(* Logix 5000 project; controller STAT 1756-L72 rev 20.12; software revision 20.04; part 10 of 34 *)
(* tags used below, declared in another part *)
   B3 : DINT[256];
   CDRO1 : REAL;
   CDRO2 : REAL;
   CDRO3 : REAL;
   COND1_EAURECYCL : REAL;
   COND2_OSMOS : DINT;
   COND3 : REAL;
   COND4 : REAL;
   COND7 : REAL;
   cond_6 : REAL;
   F8 : REAL[256];
   FLW_CO1 : REAL;
   FLW_CO2 : REAL;
   FLW_CO3 : REAL;
   FLW_EAU_VILLE : REAL;
   FLW_PO1 : REAL;
   FLW_PO2 : REAL;
   FLW_PO3 : REAL;
   hard : REAL;
   I20_000 : ALIAS FOR I20[0];
   I20_001 : ALIAS FOR I20[1];
   I20_002 : ALIAS FOR I20[2];
   I20_003 : ALIAS FOR I20[3];
   I20_004 : ALIAS FOR I20[4];
   I20_005 : ALIAS FOR I20[5];
   I20_006 : ALIAS FOR I20[6];
   I20_007 : ALIAS FOR I20[7];
   I21_000 : ALIAS FOR I21[0];
   I21_001 : ALIAS FOR I21[1];
   I21_002 : ALIAS FOR I21[2];
   I21_003 : ALIAS FOR I21[3];
   I21_004 : ALIAS FOR I21[4];
   I21_005 : ALIAS FOR I21[5];
   I21_006 : ALIAS FOR I21[6];
   I22_000 : ALIAS FOR I22[0];
   I22_001 : ALIAS FOR I22[1];
   I22_002 : ALIAS FOR I22[2];
   I22_003 : ALIAS FOR I22[3];
   I22_004 : ALIAS FOR I22[4];
   I22_005 : ALIAS FOR I22[5];
   I22_006 : ALIAS FOR I22[6];
   I22_007 : ALIAS FOR I22[7];
   I23_000 : ALIAS FOR I23[0];
   I23_001 : DINT;
   I23_003 : ALIAS FOR I23[3];
   I23_004 : ALIAS FOR I23[4];
   I23_005 : ALIAS FOR I23[5];
   I23_006 : ALIAS FOR I23[6];
   I24_000 : ALIAS FOR I24[0];
   I25_000 : ALIAS FOR I25[0];
   I25_001 : ALIAS FOR I25[1];
   I25_002 : ALIAS FOR I25[2];
   I25_003 : ALIAS FOR I25[3];
   I25_005 : ALIAS FOR I25[5];
   I25_006 : ALIAS FOR I25[6];
   I25_007 : ALIAS FOR I25[7];
   I26_000 : ALIAS FOR I26[0];
   I26_001 : ALIAS FOR I26[1];
   I26_002 : ALIAS FOR I26[2];
   int_flw_put3 : integrat;
   KRK_K1 : REAL;
   LDN_L1 : DINT;
   LVL_AZ : REAL;
   LVL_LUS2_ACIDE : REAL;
   LVL_LUS3_NAOH : REAL;
   LVL_PRETRAITEMENT : REAL;
   LVL_PUISARD_IBT : DINT;
   LVL_PUISARD_L4 : REAL;
   LVL_ZOUT : REAL;
   MW : BOOL;
   N12 : DINT[230];
   N12_110 : REAL;
   N12_14 : REAL;
   N12_38 : REAL;
   N12_44 : REAL;
   N19 : DINT[80];
   N23 : DINT[80];
   N26 : DINT[256];
   N7 : DINT[255];
   N7_70 : REAL;
   N7_72 : REAL;
   O22_000_Bit04 : ALIAS FOR O22[0].4;
   PH11 : REAL;
   PH12 : REAL;
   PH2_PRETRAIT : REAL;
   Q2 : REAL;
   Q3 : REAL;
   Q4 : REAL;
   QUAT_Q1 : REAL;
   S_FLOW_PUT_1 : DINT;
   S_FLOW_PUT_2 : DINT;
   S_FLOW_VENTURI : DINT;
   S_LVL_VIJVER : REAL;
   scp_110 : SCP;
   scp_cdro1 : SCP;
   scp_cdro2 : SCP;
   scp_cdro3 : SCP;
   scp_COND1 : SCP;
   scp_COND2_OS : SCP;
   scp_COND3 : SCP;
   scp_COND4 : SCP;
   scp_COND7 : SCP;
   scp_cond_venturi : SCP;
   scp_EAU_VILLE : SCP;
   scp_FLW_CO1 : SCP;
   scp_FLW_CO2 : SCP;
   scp_FLW_CO3 : SCP;
   scp_FLW_PO1 : SCP;
   scp_FLW_PO2 : SCP;
   scp_FLW_PO3 : SCP;
   scp_flw_put1 : SCP;
   scp_flw_put2 : SCP;
   scp_flw_put3 : SCP;
   scp_FLW_Q3 : SCP;
   scp_flw_venturi : SCP;
   scp_hard : SCP;
   scp_KR_1 : SCP;
   scp_LDN_1 : SCP;
   scp_LUS2 : SCP;
   scp_LUS3 : SCP;
   scp_LVL_AZ : SCP;
   scp_lvl_l4 : SCP;
   scp_LVL_PRET : SCP;
   scp_LVL_PUIS : SCP;
   scp_LVL_PUIS_L4 : SCP;
   scp_lvl_vijver : SCP;
   scp_LVL_ZOUT : SCP;
   scp_N12_14 : SCP;
   scp_N12_38 : SCP;
   scp_N12_44 : SCP;
   scp_N7_70 : SCP;
   scp_N7_72 : SCP;
   scp_PH11 : SCP;
   scp_PH12 : SCP;
   scp_PH2 : SCP;
   scp_ph_venturi : SCP;
   scp_Q2 : SCP;
   scp_Q4 : SCP;
   scp_QUAT_Q1 : SCP;
   scp_t_venturi : SCP;
   scpcond_6 : SCP;
(* ibt, continued *)

ROUTINE _13_ANALOG   (* ladder *)
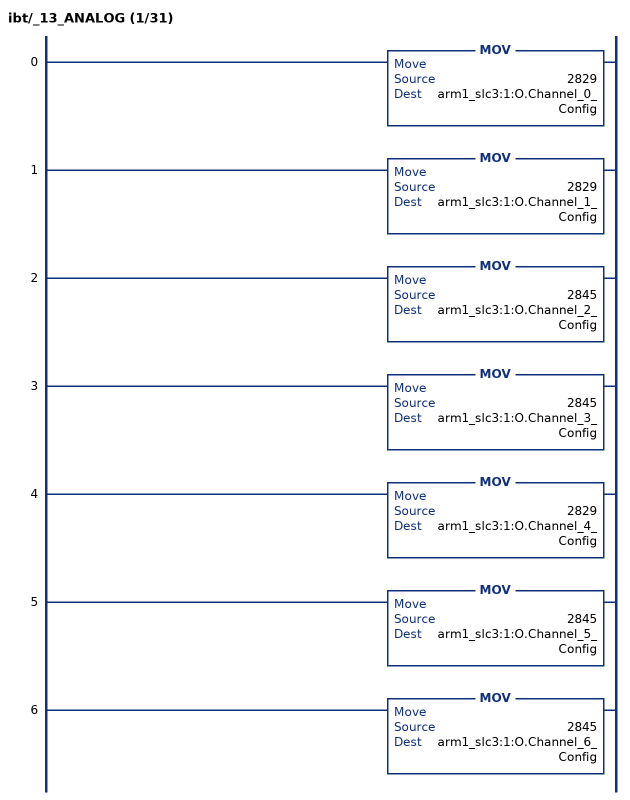
   0: MOV(2829,arm1_slc3:1:O.Channel_0_Config);
   1: MOV(2829,arm1_slc3:1:O.Channel_1_Config);
   2: MOV(2845,arm1_slc3:1:O.Channel_2_Config);
   3: MOV(2845,arm1_slc3:1:O.Channel_3_Config);
   4: MOV(2829,arm1_slc3:1:O.Channel_4_Config);
   5: MOV(2845,arm1_slc3:1:O.Channel_5_Config);
   6: MOV(2845,arm1_slc3:1:O.Channel_6_Config);
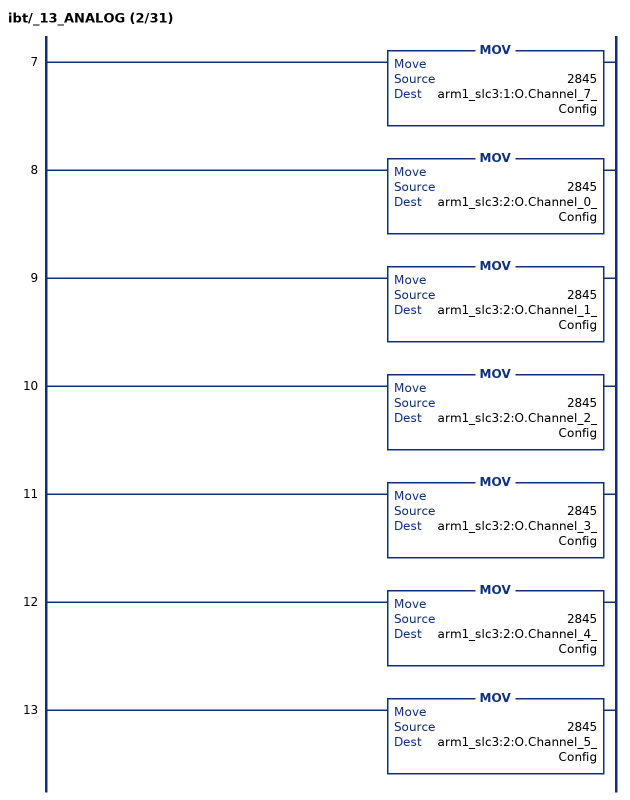
   7: MOV(2845,arm1_slc3:1:O.Channel_7_Config);
   8: MOV(2845,arm1_slc3:2:O.Channel_0_Config);
   9: MOV(2845,arm1_slc3:2:O.Channel_1_Config);
   10: MOV(2845,arm1_slc3:2:O.Channel_2_Config);
   11: MOV(2845,arm1_slc3:2:O.Channel_3_Config);
   12: MOV(2845,arm1_slc3:2:O.Channel_4_Config);
   13: MOV(2845,arm1_slc3:2:O.Channel_5_Config);
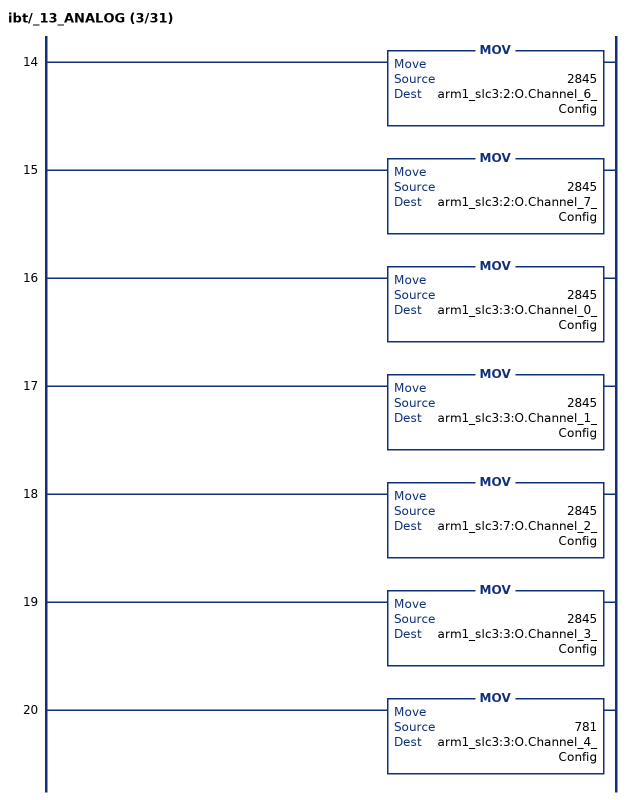
   14: MOV(2845,arm1_slc3:2:O.Channel_6_Config);
   15: MOV(2845,arm1_slc3:2:O.Channel_7_Config);
   16: MOV(2845,arm1_slc3:3:O.Channel_0_Config);
   17: MOV(2845,arm1_slc3:3:O.Channel_1_Config);
   18: MOV(2845,arm1_slc3:7:O.Channel_2_Config);
   19: MOV(2845,arm1_slc3:3:O.Channel_3_Config);
   20: MOV(781,arm1_slc3:3:O.Channel_4_Config);
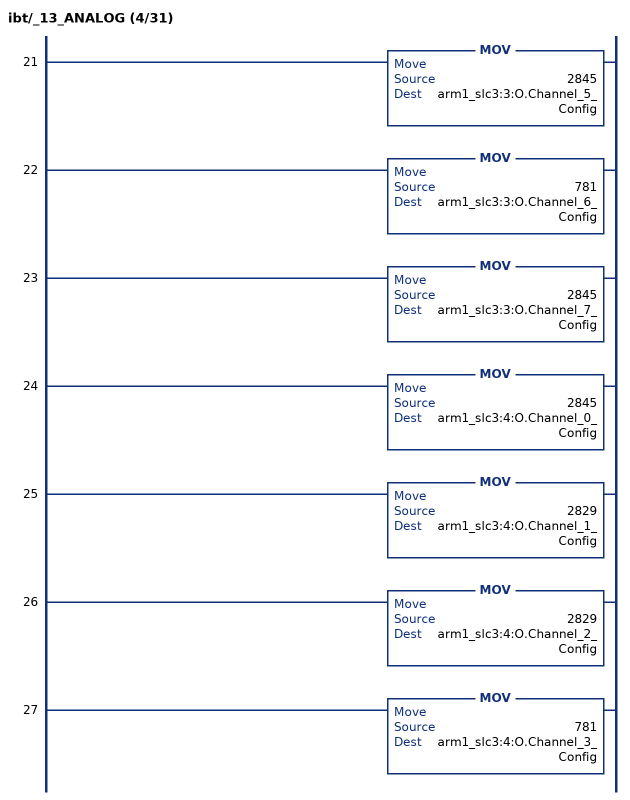
   21: MOV(2845,arm1_slc3:3:O.Channel_5_Config);
   22: MOV(781,arm1_slc3:3:O.Channel_6_Config);
   23: MOV(2845,arm1_slc3:3:O.Channel_7_Config);
   24: MOV(2845,arm1_slc3:4:O.Channel_0_Config);
   25: MOV(2829,arm1_slc3:4:O.Channel_1_Config);
   26: MOV(2829,arm1_slc3:4:O.Channel_2_Config);
   27: MOV(781,arm1_slc3:4:O.Channel_3_Config);
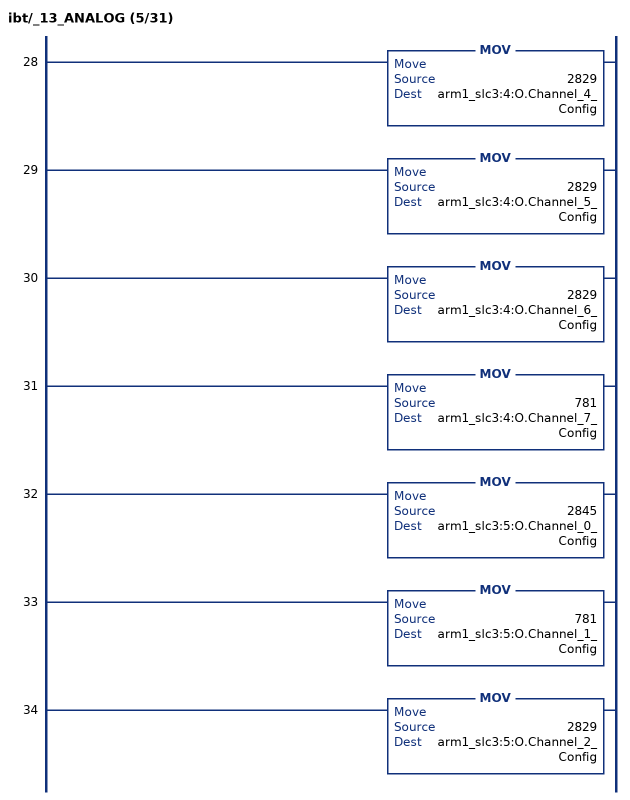
   28: MOV(2829,arm1_slc3:4:O.Channel_4_Config);
   29: MOV(2829,arm1_slc3:4:O.Channel_5_Config);
   30: MOV(2829,arm1_slc3:4:O.Channel_6_Config);
   31: MOV(781,arm1_slc3:4:O.Channel_7_Config);
   32: MOV(2845,arm1_slc3:5:O.Channel_0_Config);
   33: MOV(781,arm1_slc3:5:O.Channel_1_Config);
   34: MOV(2829,arm1_slc3:5:O.Channel_2_Config);
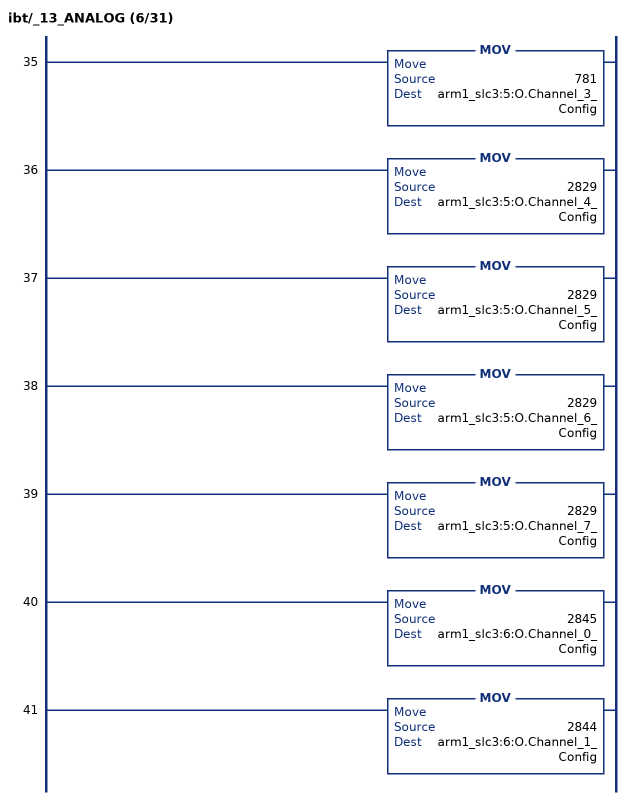
   35: MOV(781,arm1_slc3:5:O.Channel_3_Config);
   36: MOV(2829,arm1_slc3:5:O.Channel_4_Config);
   37: MOV(2829,arm1_slc3:5:O.Channel_5_Config);
   38: MOV(2829,arm1_slc3:5:O.Channel_6_Config);
   39: MOV(2829,arm1_slc3:5:O.Channel_7_Config);
   40: MOV(2845,arm1_slc3:6:O.Channel_0_Config);
   41: MOV(2844,arm1_slc3:6:O.Channel_1_Config);
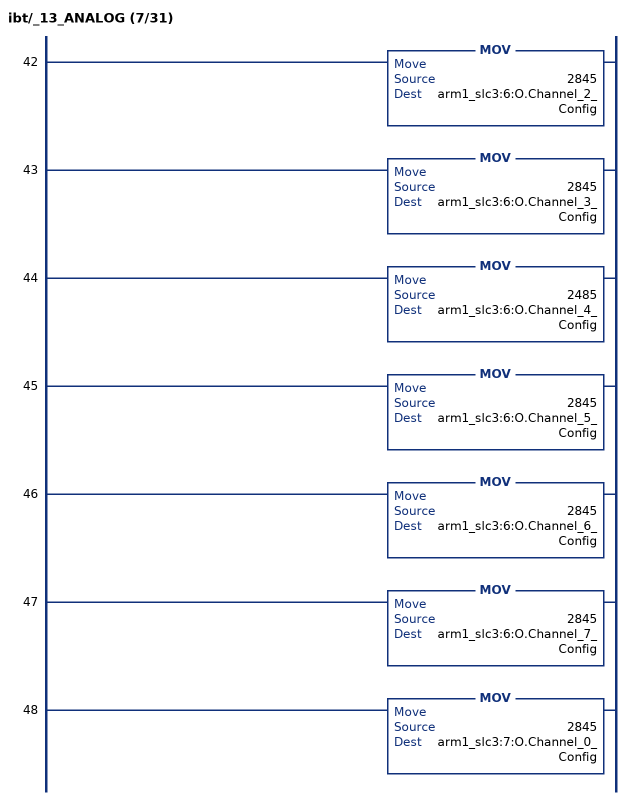
   42: MOV(2845,arm1_slc3:6:O.Channel_2_Config);
   43: MOV(2845,arm1_slc3:6:O.Channel_3_Config);
   44: MOV(2485,arm1_slc3:6:O.Channel_4_Config);
   45: MOV(2845,arm1_slc3:6:O.Channel_5_Config);
   46: MOV(2845,arm1_slc3:6:O.Channel_6_Config);
   47: MOV(2845,arm1_slc3:6:O.Channel_7_Config);
   48: MOV(2845,arm1_slc3:7:O.Channel_0_Config);
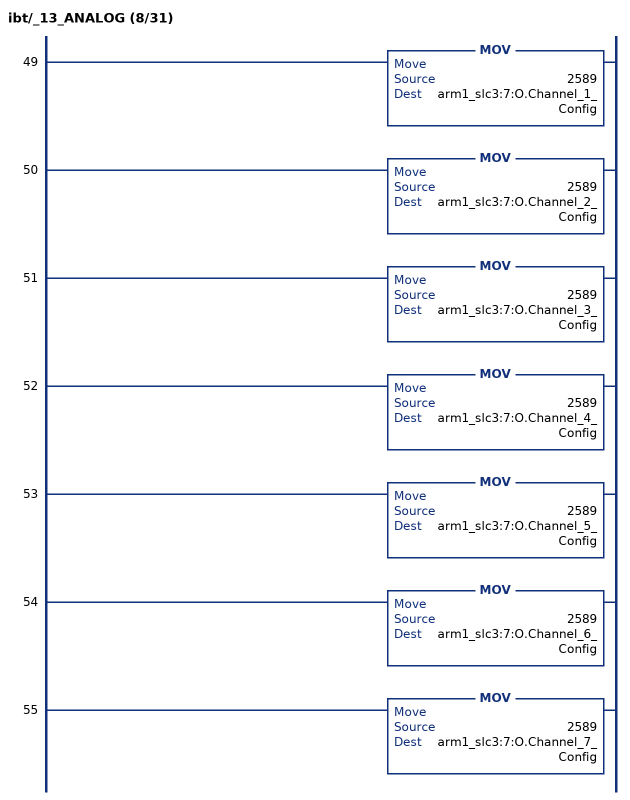
   49: MOV(2589,arm1_slc3:7:O.Channel_1_Config);
   50: MOV(2589,arm1_slc3:7:O.Channel_2_Config);
   51: MOV(2589,arm1_slc3:7:O.Channel_3_Config);
   52: MOV(2589,arm1_slc3:7:O.Channel_4_Config);
   53: MOV(2589,arm1_slc3:7:O.Channel_5_Config);
   54: MOV(2589,arm1_slc3:7:O.Channel_6_Config);
   55: MOV(2589,arm1_slc3:7:O.Channel_7_Config);
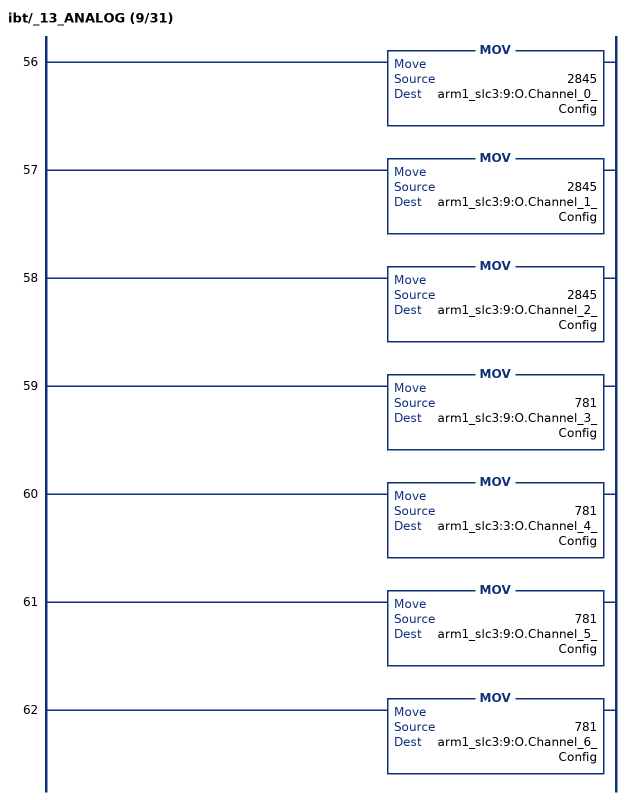
   56: MOV(2845,arm1_slc3:9:O.Channel_0_Config);
   57: MOV(2845,arm1_slc3:9:O.Channel_1_Config);
   58: MOV(2845,arm1_slc3:9:O.Channel_2_Config);
   59: MOV(781,arm1_slc3:9:O.Channel_3_Config);
   60: MOV(781,arm1_slc3:3:O.Channel_4_Config);
   61: MOV(781,arm1_slc3:9:O.Channel_5_Config);
   62: MOV(781,arm1_slc3:9:O.Channel_6_Config);
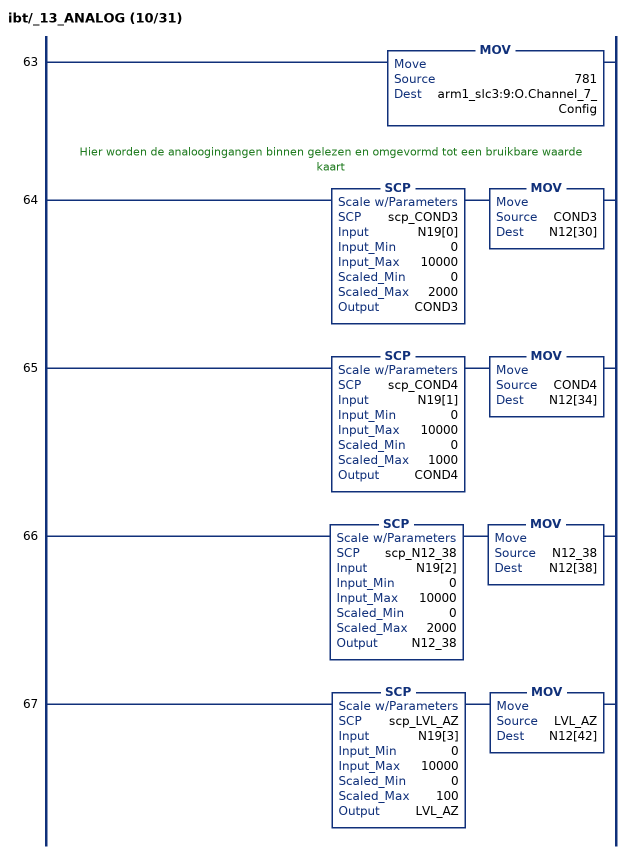
   63: MOV(781,arm1_slc3:9:O.Channel_7_Config);
   // Hier worden de analoogingangen binnen gelezen en omgevormd tot een bruikbare waarde kaart
   64: SCP(scp_COND3,N19[0],0,10000,0,2000,COND3)MOV(COND3,N12[30]);
   65: SCP(scp_COND4,N19[1],0,10000,0,1000,COND4)MOV(COND4,N12[34]);
   66: SCP(scp_N12_38,N19[2],0,10000,0,2000,N12_38)MOV(N12_38,N12[38]);
   67: SCP(scp_LVL_AZ,N19[3],0,10000,0,100,LVL_AZ)MOV(LVL_AZ,N12[42]);
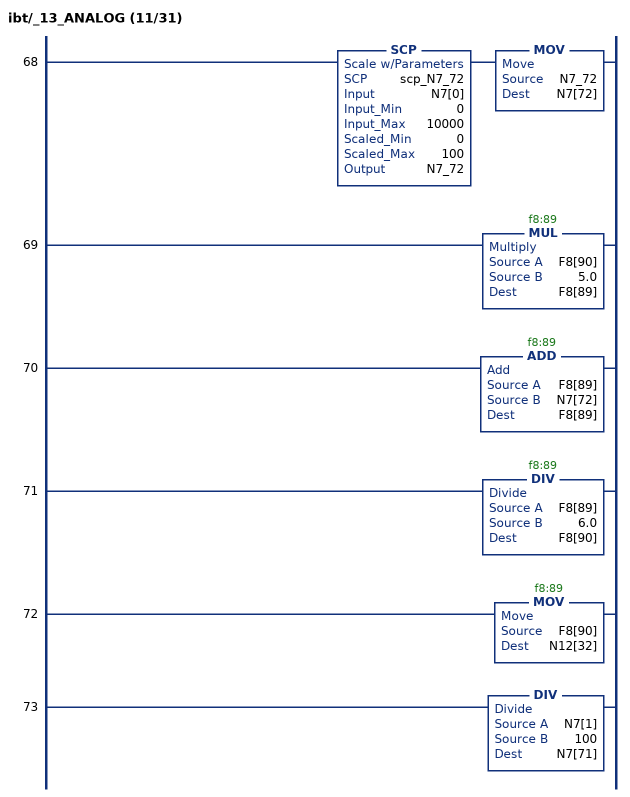
   68: SCP(scp_N7_72,N7[0],0,10000,0,100,N7_72)MOV(N7_72,N7[72]);
   69: MUL(F8[90],5.0,F8[89]);
   70: ADD(F8[89],N7[72],F8[89]);
   71: DIV(F8[89],6.0,F8[90]);
   72: MOV(F8[90],N12[32]);
   73: DIV(N7[1],100,N7[71]);
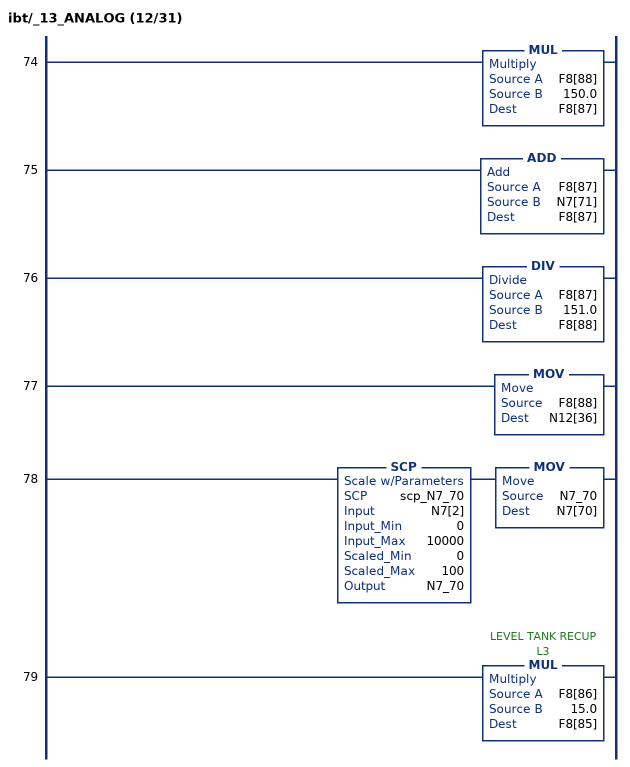
   74: MUL(F8[88],150.0,F8[87]);
   75: ADD(F8[87],N7[71],F8[87]);
   76: DIV(F8[87],151.0,F8[88]);
   77: MOV(F8[88],N12[36]);
   78: SCP(scp_N7_70,N7[2],0,10000,0,100,N7_70)MOV(N7_70,N7[70]);
   79: MUL(F8[86],15.0,F8[85]);
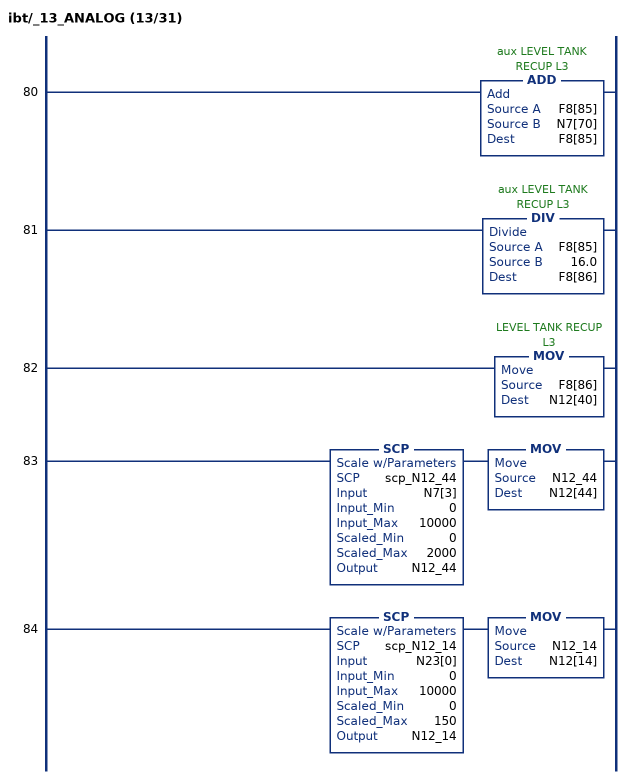
   80: ADD(F8[85],N7[70],F8[85]);
   81: DIV(F8[85],16.0,F8[86]);
   82: MOV(F8[86],N12[40]);
   83: SCP(scp_N12_44,N7[3],0,10000,0,2000,N12_44)MOV(N12_44,N12[44]);
   84: SCP(scp_N12_14,N23[0],0,10000,0,150,N12_14)MOV(N12_14,N12[14]);
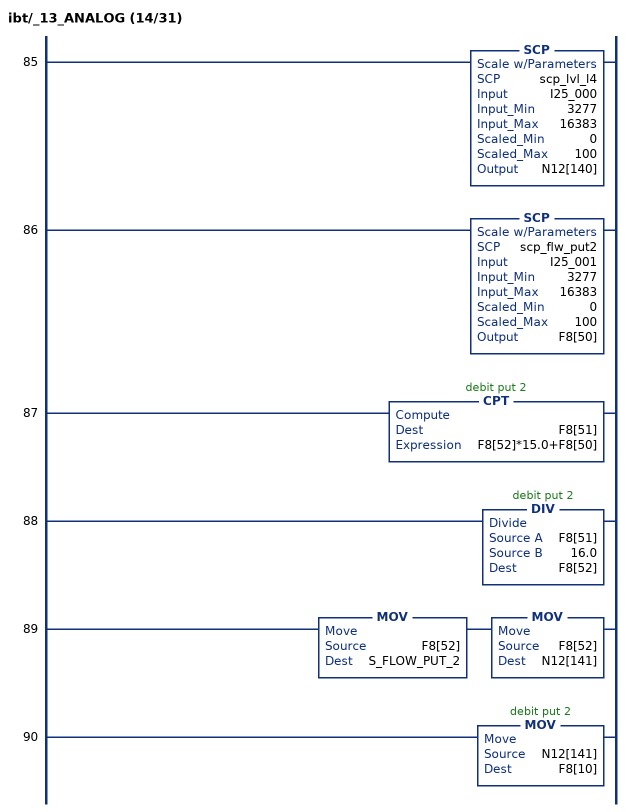
   85: SCP(scp_lvl_l4,I25_000,3277,16383,0,100,N12[140]);
   86: SCP(scp_flw_put2,I25_001,3277,16383,0,100,F8[50]);
   87: CPT(F8[51],F8[52]*15.0+F8[50]);
   88: DIV(F8[51],16.0,F8[52]);
   89: MOV(F8[52],S_FLOW_PUT_2)MOV(F8[52],N12[141]);
   90: MOV(N12[141],F8[10]);
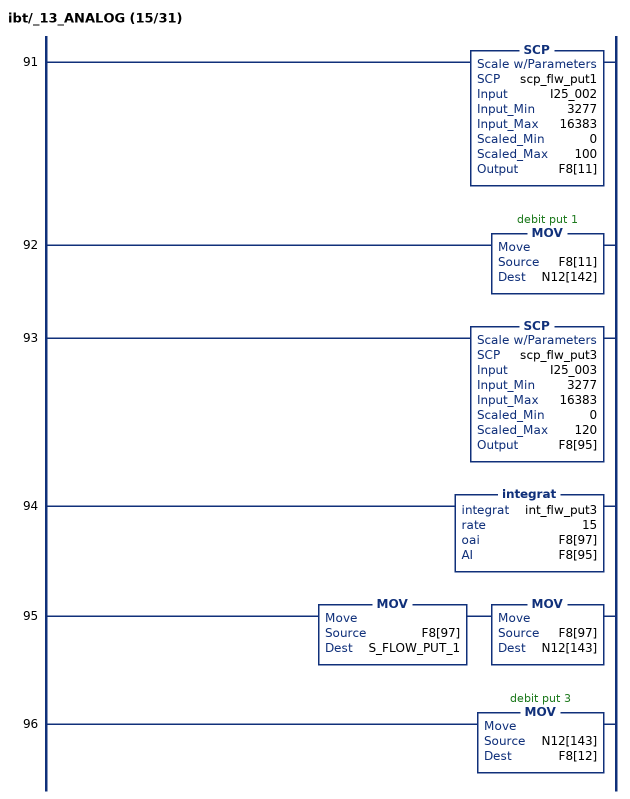
   91: SCP(scp_flw_put1,I25_002,3277,16383,0,100,F8[11]);
   92: MOV(F8[11],N12[142]);
   93: SCP(scp_flw_put3,I25_003,3277,16383,0,120,F8[95]);
   94: integrat(int_flw_put3,15,F8[97],F8[95]);
   95: MOV(F8[97],S_FLOW_PUT_1)MOV(F8[97],N12[143]);
   96: MOV(N12[143],F8[12]);
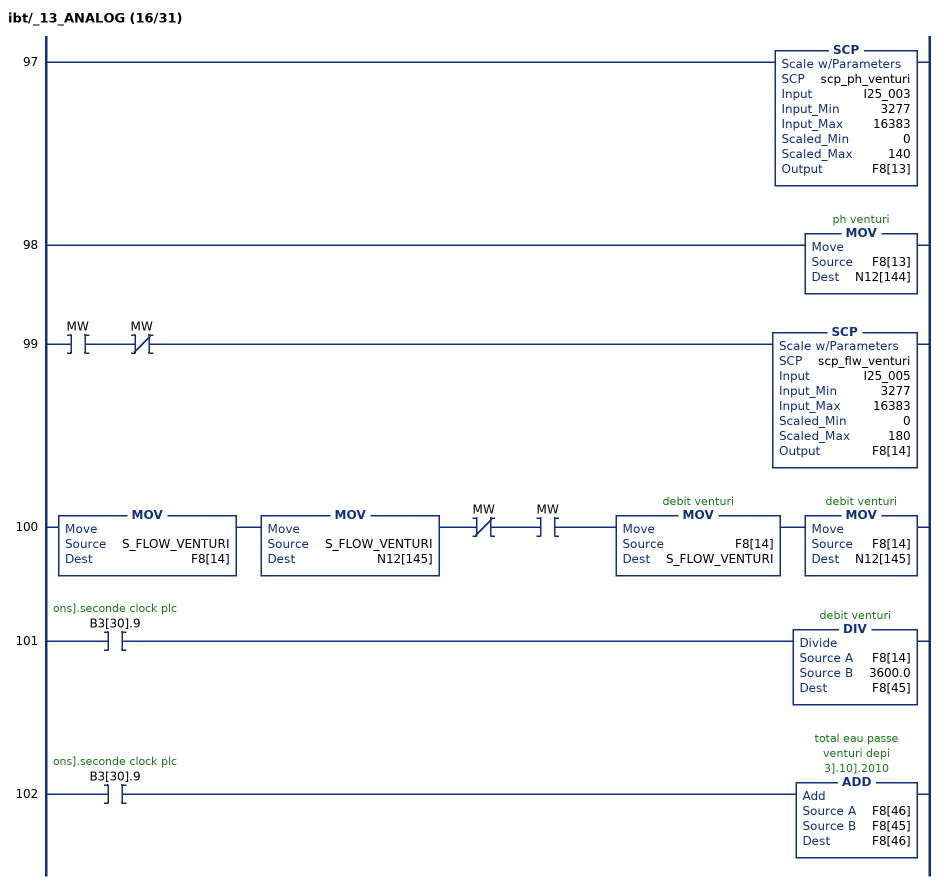
   97: SCP(scp_ph_venturi,I25_003,3277,16383,0,140,F8[13]);
   98: MOV(F8[13],N12[144]);
   99: XIC(MW)XIO(MW)SCP(scp_flw_venturi,I25_005,3277,16383,0,180,F8[14]);
   100: MOV(S_FLOW_VENTURI,F8[14])MOV(S_FLOW_VENTURI,N12[145])XIO(MW)XIC(MW)MOV(F8[14],S_FLOW_VENTURI)MOV(F8[14],N12[145]);
   101: XIC(B3[30].9)DIV(F8[14],3600.0,F8[45]);
   102: XIC(B3[30].9)ADD(F8[46],F8[45],F8[46]);
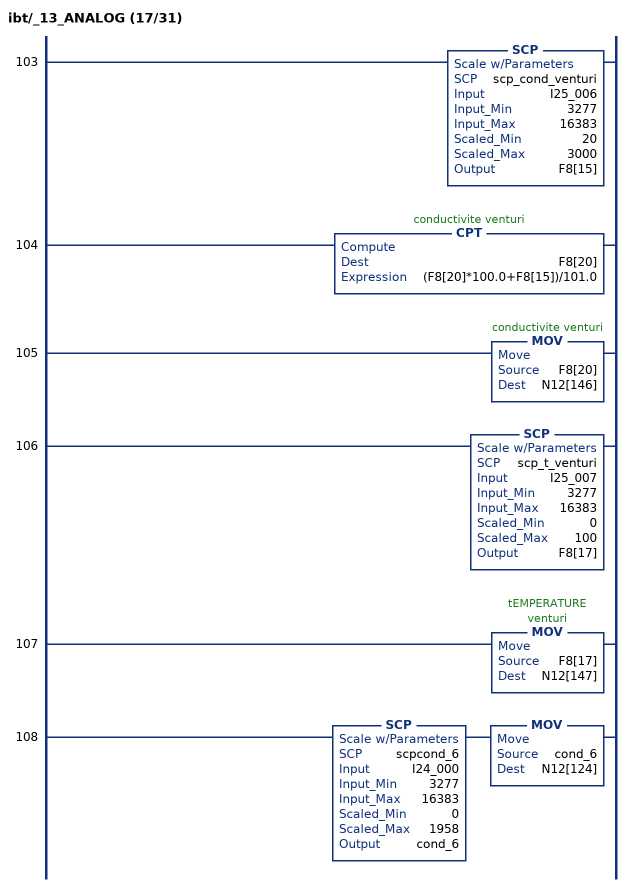
   103: SCP(scp_cond_venturi,I25_006,3277,16383,20,3000,F8[15]);
   104: CPT(F8[20],(F8[20]*100.0+F8[15])/101.0);
   105: MOV(F8[20],N12[146]);
   106: SCP(scp_t_venturi,I25_007,3277,16383,0,100,F8[17]);
   107: MOV(F8[17],N12[147]);
   108: SCP(scpcond_6,I24_000,3277,16383,0,1958,cond_6)MOV(cond_6,N12[124]);
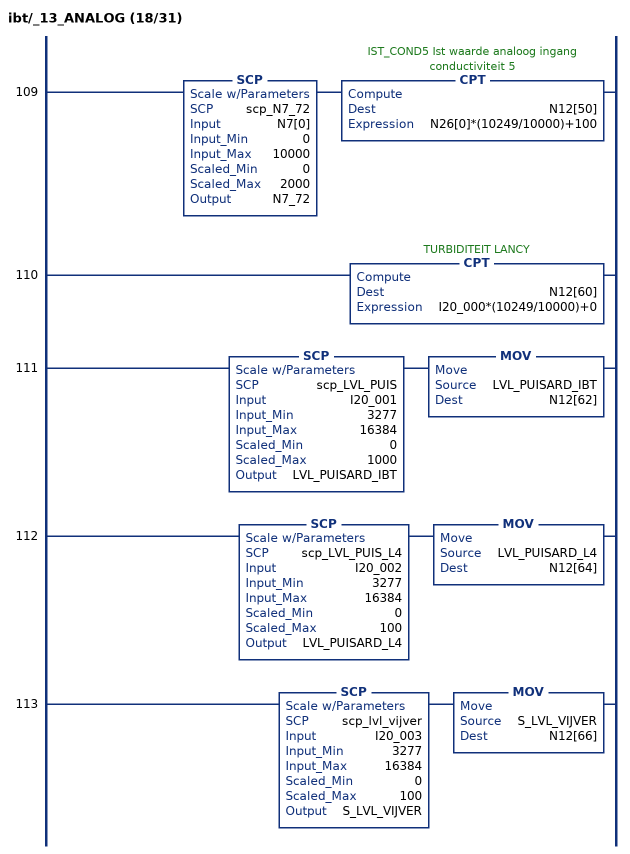
   109: SCP(scp_N7_72,N7[0],0,10000,0,2000,N7_72)CPT(N12[50],N26[0]*(10249/10000)+100);
   110: CPT(N12[60],I20_000*(10249/10000)+0);
   111: SCP(scp_LVL_PUIS,I20_001,3277,16384,0,1000,LVL_PUISARD_IBT)MOV(LVL_PUISARD_IBT,N12[62]);
   112: SCP(scp_LVL_PUIS_L4,I20_002,3277,16384,0,100,LVL_PUISARD_L4)MOV(LVL_PUISARD_L4,N12[64]);
   113: SCP(scp_lvl_vijver,I20_003,3277,16384,0,100,S_LVL_VIJVER)MOV(S_LVL_VIJVER,N12[66]);
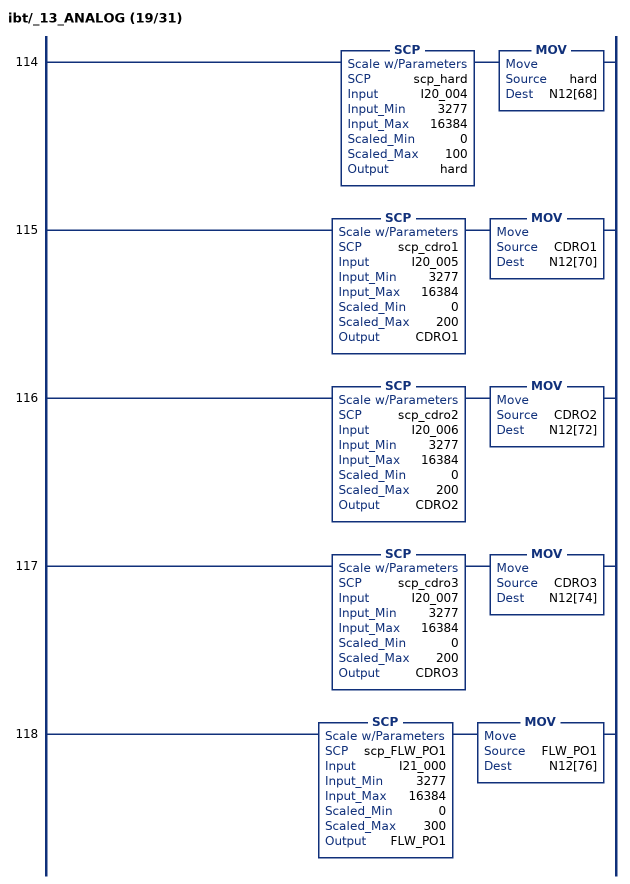
   114: SCP(scp_hard,I20_004,3277,16384,0,100,hard)MOV(hard,N12[68]);
   115: SCP(scp_cdro1,I20_005,3277,16384,0,200,CDRO1)MOV(CDRO1,N12[70]);
   116: SCP(scp_cdro2,I20_006,3277,16384,0,200,CDRO2)MOV(CDRO2,N12[72]);
   117: SCP(scp_cdro3,I20_007,3277,16384,0,200,CDRO3)MOV(CDRO3,N12[74]);
   118: SCP(scp_FLW_PO1,I21_000,3277,16384,0,300,FLW_PO1)MOV(FLW_PO1,N12[76]);
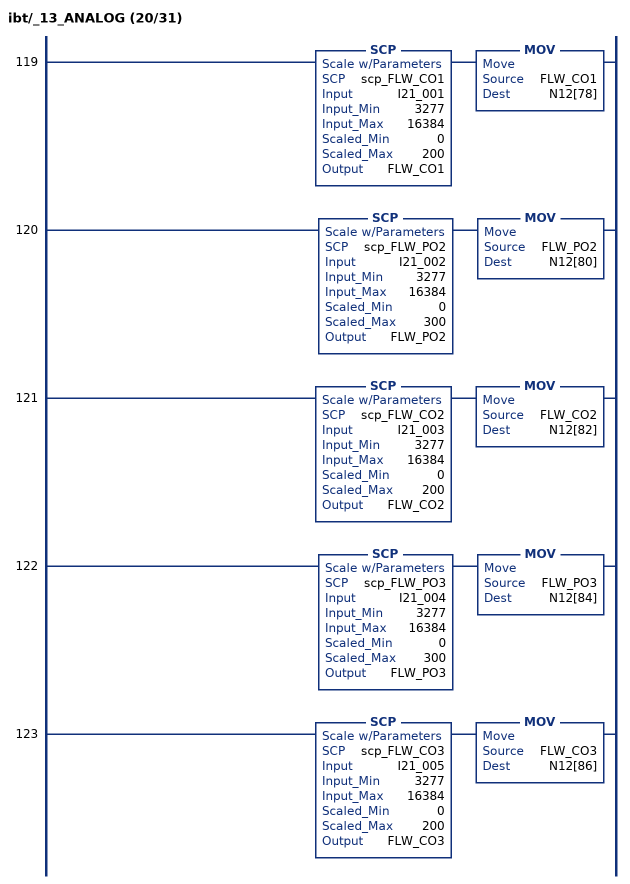
   119: SCP(scp_FLW_CO1,I21_001,3277,16384,0,200,FLW_CO1)MOV(FLW_CO1,N12[78]);
   120: SCP(scp_FLW_PO2,I21_002,3277,16384,0,300,FLW_PO2)MOV(FLW_PO2,N12[80]);
   121: SCP(scp_FLW_CO2,I21_003,3277,16384,0,200,FLW_CO2)MOV(FLW_CO2,N12[82]);
   122: SCP(scp_FLW_PO3,I21_004,3277,16384,0,300,FLW_PO3)MOV(FLW_PO3,N12[84]);
   123: SCP(scp_FLW_CO3,I21_005,3277,16384,0,200,FLW_CO3)MOV(FLW_CO3,N12[86]);
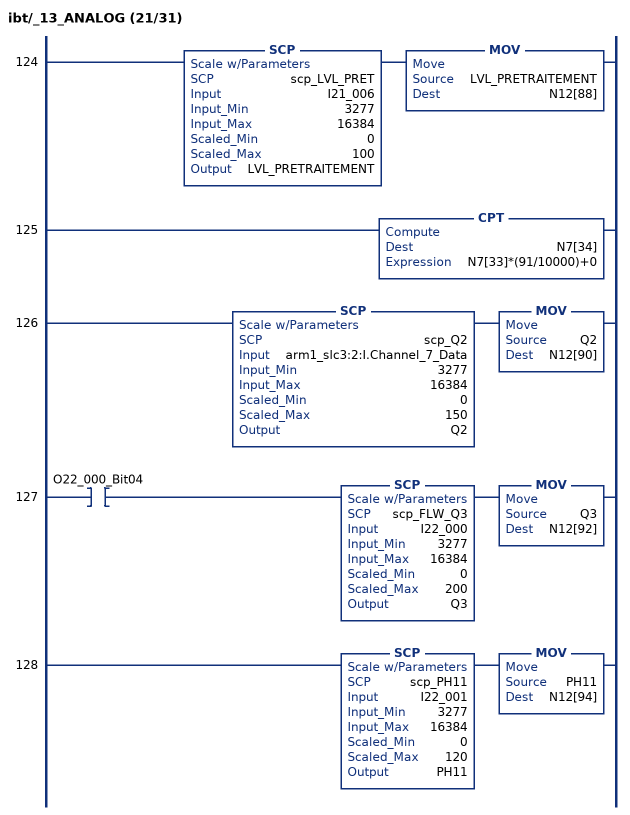
   124: SCP(scp_LVL_PRET,I21_006,3277,16384,0,100,LVL_PRETRAITEMENT)MOV(LVL_PRETRAITEMENT,N12[88]);
   125: CPT(N7[34],N7[33]*(91/10000)+0);
   126: SCP(scp_Q2,arm1_slc3:2:I.Channel_7_Data,3277,16384,0,150,Q2)MOV(Q2,N12[90]);
   127: XIC(O22_000_Bit04)SCP(scp_FLW_Q3,I22_000,3277,16384,0,200,Q3)MOV(Q3,N12[92]);
   128: SCP(scp_PH11,I22_001,3277,16384,0,120,PH11)MOV(PH11,N12[94]);
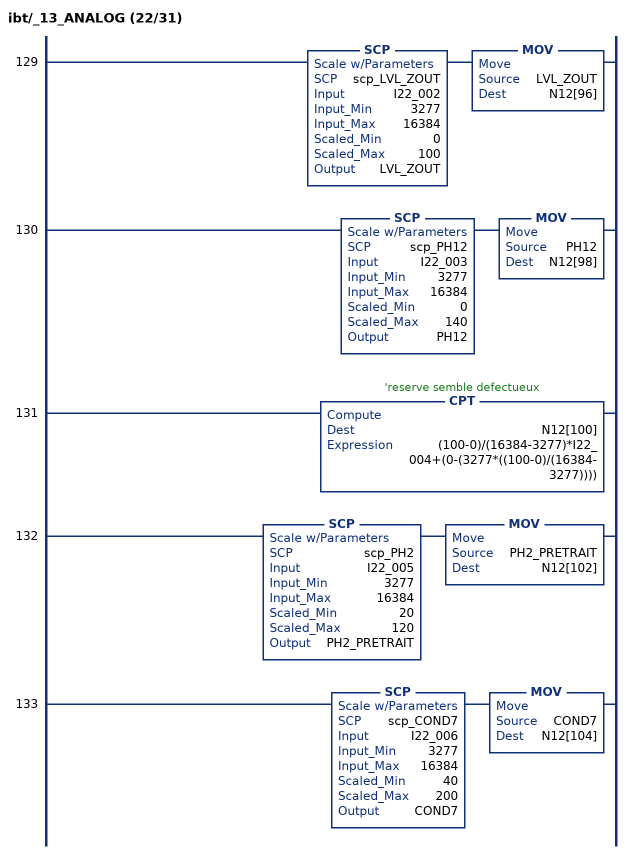
   129: SCP(scp_LVL_ZOUT,I22_002,3277,16384,0,100,LVL_ZOUT)MOV(LVL_ZOUT,N12[96]);
   130: SCP(scp_PH12,I22_003,3277,16384,0,140,PH12)MOV(PH12,N12[98]);
   131: CPT(N12[100],(100-0)/(16384-3277)*I22_004+(0-(3277*((100-0)/(16384-3277)))));
   132: SCP(scp_PH2,I22_005,3277,16384,20,120,PH2_PRETRAIT)MOV(PH2_PRETRAIT,N12[102]);
   133: SCP(scp_COND7,I22_006,3277,16384,40,200,COND7)MOV(COND7,N12[104]);
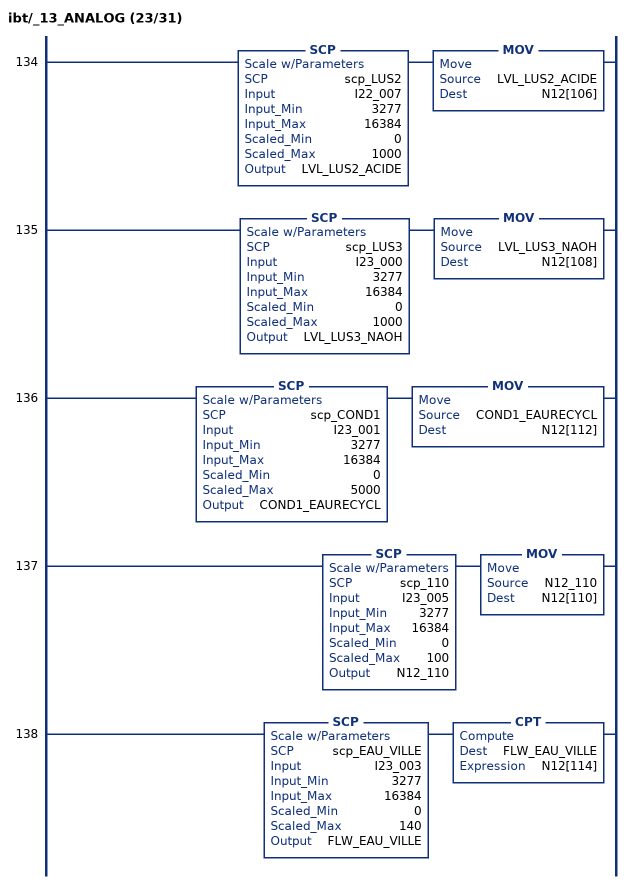
   134: SCP(scp_LUS2,I22_007,3277,16384,0,1000,LVL_LUS2_ACIDE)MOV(LVL_LUS2_ACIDE,N12[106]);
   135: SCP(scp_LUS3,I23_000,3277,16384,0,1000,LVL_LUS3_NAOH)MOV(LVL_LUS3_NAOH,N12[108]);
   136: SCP(scp_COND1,I23_001,3277,16384,0,5000,COND1_EAURECYCL)MOV(COND1_EAURECYCL,N12[112]);
   137: SCP(scp_110,I23_005,3277,16384,0,100,N12_110)MOV(N12_110,N12[110]);
   138: SCP(scp_EAU_VILLE,I23_003,3277,16384,0,140,FLW_EAU_VILLE)CPT(FLW_EAU_VILLE,N12[114]);
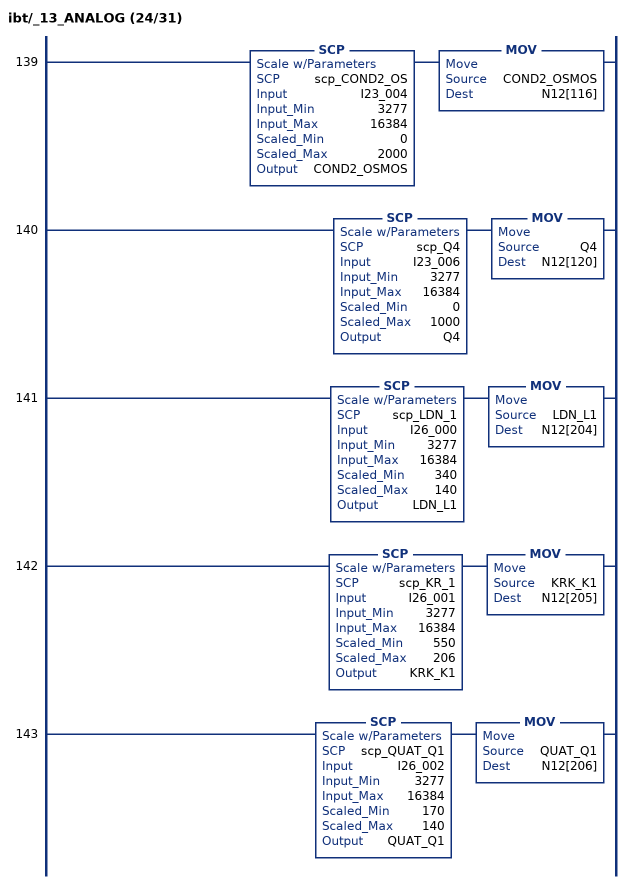
   139: SCP(scp_COND2_OS,I23_004,3277,16384,0,2000,COND2_OSMOS)MOV(COND2_OSMOS,N12[116]);
   140: SCP(scp_Q4,I23_006,3277,16384,0,1000,Q4)MOV(Q4,N12[120]);
   141: SCP(scp_LDN_1,I26_000,3277,16384,340,140,LDN_L1)MOV(LDN_L1,N12[204]);
   142: SCP(scp_KR_1,I26_001,3277,16384,550,206,KRK_K1)MOV(KRK_K1,N12[205]);
   143: SCP(scp_QUAT_Q1,I26_002,3277,16384,170,140,QUAT_Q1)MOV(QUAT_Q1,N12[206]);
